// Mitsubishi GX Works2 project: 시퀀스 예제 2   PLC: Q03UDV

PROGRAM MAIN
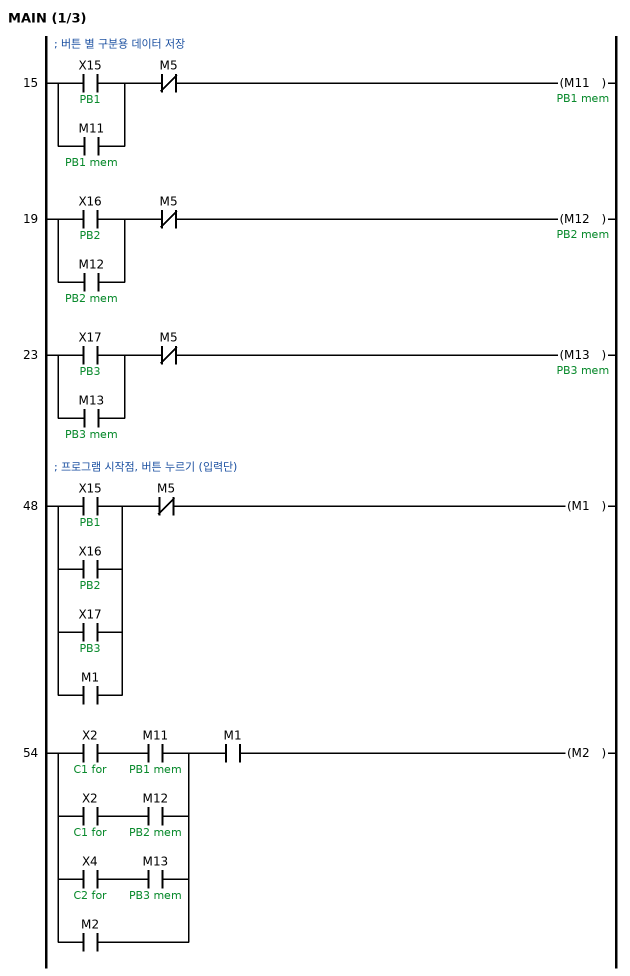
; 버튼 별 구분용 데이터 저장
15    LD      X15  ; PB1
      OR      M11  ; PB1 mem
      ANI     M5
      OUT     M11  ; PB1 mem
19    LD      X16  ; PB2
      OR      M12  ; PB2 mem
      ANI     M5
      OUT     M12  ; PB2 mem
23    LD      X17  ; PB3
      OR      M13  ; PB3 mem
      ANI     M5
      OUT     M13  ; PB3 mem
; 프로그램 시작점, 버튼 누르기 (입력단)
48    LD      X15  ; PB1
      OR      X16  ; PB2
      OR      X17  ; PB3
      OR      M1
      ANI     M5
      OUT     M1
54    LD      X2  ; C1 for
      AND     M11  ; PB1 mem
      LD      X2  ; C1 for
      AND     M12  ; PB2 mem
      ORB
      LD      X4  ; C2 for
      AND     M13  ; PB3 mem
      ORB
      OR      M2
      AND     M1
      OUT     M2
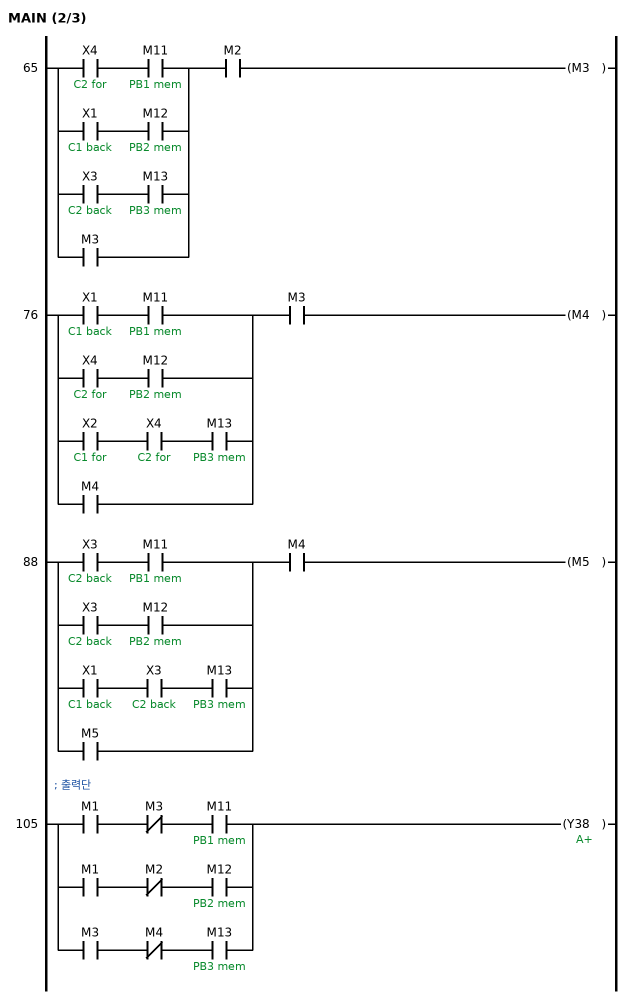
65    LD      X4  ; C2 for
      AND     M11  ; PB1 mem
      LD      X1  ; C1 back
      AND     M12  ; PB2 mem
      ORB
      LD      X3  ; C2 back
      AND     M13  ; PB3 mem
      ORB
      OR      M3
      AND     M2
      OUT     M3
76    LD      X1  ; C1 back
      AND     M11  ; PB1 mem
      LD      X4  ; C2 for
      AND     M12  ; PB2 mem
      ORB
      LD      X2  ; C1 for
      AND     X4  ; C2 for
      AND     M13  ; PB3 mem
      ORB
      OR      M4
      AND     M3
      OUT     M4
88    LD      X3  ; C2 back
      AND     M11  ; PB1 mem
      LD      X3  ; C2 back
      AND     M12  ; PB2 mem
      ORB
      LD      X1  ; C1 back
      AND     X3  ; C2 back
      AND     M13  ; PB3 mem
      ORB
      OR      M5
      AND     M4
      OUT     M5
; 출력단
105   LD      M1
      ANI     M3
      AND     M11  ; PB1 mem
      LD      M1
      ANI     M2
      AND     M12  ; PB2 mem
      ORB
      LD      M3
      ANI     M4
      AND     M13  ; PB3 mem
      ORB
      OUT     Y38  ; A+
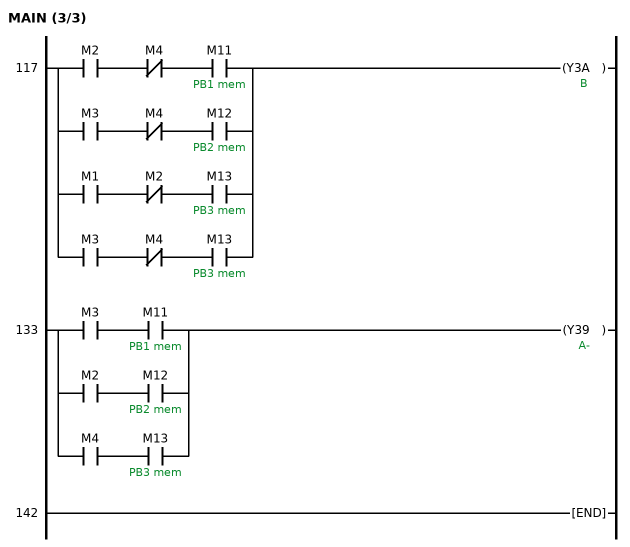
117   LD      M2
      ANI     M4
      AND     M11  ; PB1 mem
      LD      M3
      ANI     M4
      AND     M12  ; PB2 mem
      ORB
      LD      M1
      ANI     M2
      AND     M13  ; PB3 mem
      ORB
      LD      M3
      ANI     M4
      AND     M13  ; PB3 mem
      ORB
      OUT     Y3A  ; B
133   LD      M3
      AND     M11  ; PB1 mem
      LD      M2
      AND     M12  ; PB2 mem
      ORB
      LD      M4
      AND     M13  ; PB3 mem
      ORB
      OUT     Y39  ; A-
142   END
END_PROGRAM
